KUKA KRL data list: $config.dat

&ACCESS RV$3
DEFDAT $CONFIG

ENDDAT
